SUBAPPLICATION Uebung_028 (* Analog-Eingang *)
  (* Standard: 61499-2; Description: Copyright (c) 2023 Meisterschulen am Ostbahnhof This program and the accompanying materials are made available under the terms of the Eclipse Public License 2.0 which is available at https://www.eclipse.org/legal/epl-2.0/ SPDX-License-Identifier: EPL-2.0 *)
  (* Version 1.0, 2023-10-23, Franz Höpfinger, Meisterschulen am Ostbahnhof, initial API and implementation and/or initial documentation *)
  PACKAGE Uebungen;
  IMPORT logiBUS::io::DI::logiBUS_DI::Input_I1;
  IMPORT logiBUS::io::DQ::logiBUS_DO::Output_Q1;
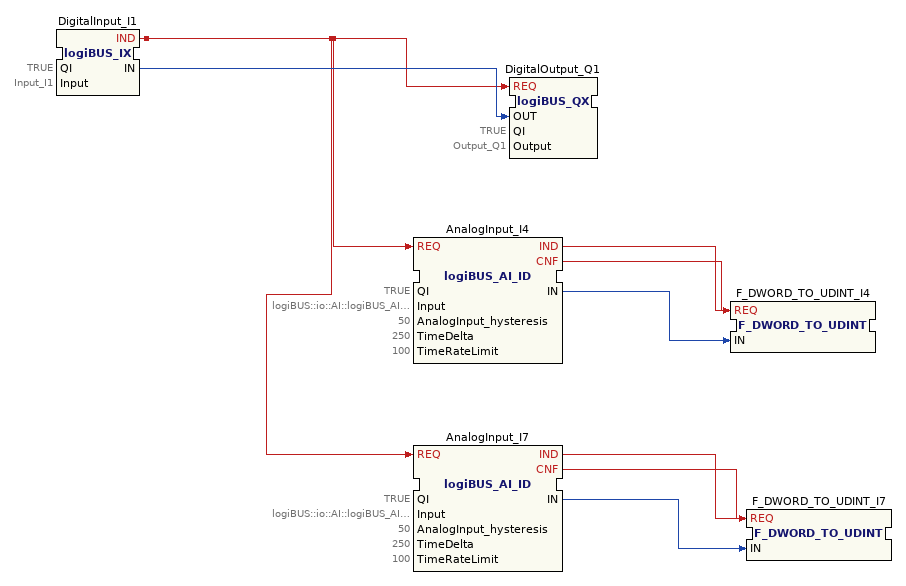
  FBS
    DigitalOutput_Q1 : logiBUS::io::DQ::logiBUS_QX(QI := TRUE, Output := Output_Q1);
    DigitalInput_I1 : logiBUS::io::DI::logiBUS_IX(QI := TRUE, Input := Input_I1);
    AnalogInput_I4 : logiBUS::io::AI::logiBUS_AI_ID(QI := TRUE, Input := logiBUS::io::AI::logiBUS_AI::AnalogInput_I4, AnalogInput_hysteresis := 50, TimeDelta := 250, TimeRateLimit := 100);
    AnalogInput_I7 : logiBUS::io::AI::logiBUS_AI_ID(QI := TRUE, Input := logiBUS::io::AI::logiBUS_AI::AnalogInput_I7, AnalogInput_hysteresis := 50, TimeDelta := 250, TimeRateLimit := 100);
    F_DWORD_TO_UDINT_I7 : iec61131::conversion::F_DWORD_TO_UDINT;
    F_DWORD_TO_UDINT_I4 : iec61131::conversion::F_DWORD_TO_UDINT;
  END_FBS
  EVENT_CONNECTIONS
    DigitalInput_I1.IND TO DigitalOutput_Q1.REQ;
    AnalogInput_I7.IND TO F_DWORD_TO_UDINT_I7.REQ;
    AnalogInput_I4.IND TO F_DWORD_TO_UDINT_I4.REQ;
    DigitalInput_I1.IND TO AnalogInput_I4.REQ;
    DigitalInput_I1.IND TO AnalogInput_I7.REQ;
    AnalogInput_I7.CNF TO F_DWORD_TO_UDINT_I7.REQ;
    AnalogInput_I4.CNF TO F_DWORD_TO_UDINT_I4.REQ;
  END_CONNECTIONS
  DATA_CONNECTIONS
    DigitalInput_I1.IN TO DigitalOutput_Q1.OUT;
    AnalogInput_I7.IN TO F_DWORD_TO_UDINT_I7.IN;
    AnalogInput_I4.IN TO F_DWORD_TO_UDINT_I4.IN;
  END_CONNECTIONS
END_SUBAPPLICATION
